// TIA Portal V19 export
TYPE "EFC_EX_STATUS_WORD"
   STRUCT
      Reserved0 : Bool := false;
      Reserved1 : Bool := false;
      Reserved2 : Bool := false;
      Reserved3 : Bool := false;
      Reserved4 : Bool := false;
      Reserved5 : Bool := false;
      Warning : Bool := false;
      Reserved7 : Bool := false;
      Mode24V : Bool := false;
      SleepMode : Bool := false;
      ConverterOk : Bool := false;
      Reserved11 : Bool := false;
      Reserved12 : Bool := false;
      Reserved13 : Bool := false;
      Reserved14 : Bool := false;
      Reserved15 : Bool := false;
   END_STRUCT;
END_TYPE
